{attribute 'linkalways'}
{attribute 'hide_all_locals'}
FUNCTION_BLOCK ValueUsint EXTENDS ValueUsintRead IMPLEMENTS Value
VAR
END_VAR

METHOD SetFromType : BOOL
VAR_INPUT
	source : __SYSTEM.AnyType;
END_VAR
SetFromType := ConvertAnyType(source, thisAnyType);
END_METHOD

METHOD SetFromString : BOOL
VAR_INPUT
	value : T_MaxString;
END_VAR
thisValue := STRING_TO_USINT(value);

SetFromString := TRUE;
END_METHOD

METHOD Set : BOOL
VAR_INPUT
	source : ANY;
END_VAR
Set := ConvertAnyType(source, thisAnyType);
END_METHOD

END_FUNCTION_BLOCK

(* stored: Version 1.1.0.1
   POU ValueUsint: Id {02404ce2-8b87-419e-957f-e4f3a2e57a24}, SpecialFunc None
   Method SetFromType: Id {156d6418-133f-4bf7-a9c6-ff9607901626}
   Method SetFromString: Id {87ce5a61-e4e9-4326-92e7-a9c03a5bb114}
   Method Set: Id {144ff643-873b-4125-bea3-f44b3d27aa5f} *)
